Fanuc KAREL source: ko00094.KL

-- PROVISIONAL review KL for V770-1; original PC SHA256 9dd6879cb9382386aa4a65f620fbd0d1322e37865e86d95fa055d886a99c3e6c
-- Incomplete behavior may be omitted. Consult companion uncertainty JSON. Do not deploy.
PROGRAM KO00094
%NOLOCKGROUP
BEGIN
  -- UNRESOLVED_PC offsets 5-12; opcodes 9D,23
  -- UNRESOLVED_PC offsets 17-69; opcodes 27,27,49,7E,AD,27,49,7E,AD,22,31,7E,4A
  -- UNRESOLVED_PC offsets 74-78; opcodes 7F
END KO00094
